(* CoDeSys 2.3.9.47 project: derevo_2016_12_28.pr6 *)
(* Author: Yurko Shybaigolova *)
(* Libraries: PlcHelperBC.lb6 7.5.01 11:03:00, TcAdsBC.lb6 5.7.02 11:03:02, standard.lb6 5.6.98 11:03:02, PlcSystemBC.lb6 21.3.01 11:03:02, TcBABasicBC.lb6 22.7.15 15:46:36, TcPlcUtilitiesBC.lb6 13.5.05 11:19:40 *)

(* Global variable list: main *)
VAR_GLOBAL
	data3floor: ARRAY[0..100] OF BYTE;
	data3floor_prev :ARRAY[0..100] OF BYTE;

	ads_adr1: STRING:='10.0.5.61.1.1';
	ads_adr2: STRING:='10.0.5.62.1.1';
	ads_adr3: STRING:='10.0.5.63.1.1';
	ads_adr_gym: STRING:='10.0.5.67.1.1';

	write_ads: ADSWRITE;
	basseinWindowToSafePos: BOOL;

	bDarkOutside		AT%MX0.0:BOOL;


	iHour			AT%MB4:BYTE;
	iMinute			AT%MB5:BYTE;
	lights			AT%MB6:DWORD;
	t_out			AT%MB10:INT;

	eib_vidpochynok1 				AT %MX100.0:	 BOOL;
	eib_vidpochynok2 				AT %MX100.1:	 BOOL;
	eib_veranda 					AT %MX100.2:	 BOOL;
	eib_veranda_zovn 				AT %MX100.3:	 BOOL;
	eib_vhid_zovn 					AT %MX100.4:	 BOOL;
	eib_sauna 						AT %MX100.5:	 BOOL;
	eib_vhid						AT %MX100.6:	 BOOL;
	eib_kotel 						AT %MX100.7:	 BOOL;

	eib_korydor 						AT %MX101.0:	 BOOL;
	eib_sinna 						AT %MX101.1:	 BOOL;
	eib_hamam 						AT %MX101.2:	 BOOL;
	eib_kuhnya 						AT %MX101.3:	 BOOL;
	eib_bassein1					AT %MX101.4:	 BOOL;
	eib_bassein_lampa				AT %MX101.5:	 BOOL;
	eib_spalnya2					AT %MX101.6:	 BOOL;
	eib_terassa 						AT %MX101.7:	 BOOL;

	eib_dush 						AT %MX102.0:	 BOOL;
	eib_wc 							AT %MX102.1:	 BOOL;
	eib_spalnya_verh				AT %MX102.2:	 BOOL;
	eib_spalnya1 					AT %MX102.3:	 BOOL;
	eib_spalnya_su 					AT %MX102.4:	 BOOL;
	eib_garderob 					AT %MX102.5:	 BOOL;
	eib_dush2						AT %MX102.6:	 BOOL;

	eib_okno_basseina				AT %MX103.0:	 BOOL;

	okno_basseina_status: BOOL;

	dataToGym0					AT %MB105: 	 BYTE;
	dataToGym1					AT %MB106: 	 BYTE;
	dataToGym2					AT %MB107: 	 BYTE;
	dataToGym3					AT %MB108: 	 BYTE;
	dataToGym4					AT %MB109: 	 BYTE;
	dataToGym5					AT %MB110: 	 BYTE;
	dataToGym6					AT %MB111: 	 BYTE;
	dataToGym7					AT %MB112: 	 BYTE;
	dataToGym8					AT %MB113: 	 BYTE;

	dataFromGym 				AT %MB300:	ARRAY[0..15] OF BYTE;





END_VAR

(* Global variable list: physical *)
(* @GLOBAL_VARIABLE_LIST := TwinCAT_Import *)
(* @PATH := '' *)
VAR_GLOBAL (* DO NOT CHANGE THIS SHEET MANUALLY! *)
	PlcInVar_0	AT %QB128:	USINT;
	PlcInVar_1	AT %QB129:	USINT;
	PlcInVar_2	AT %QB130:	USINT;
	PlcInVar_3	AT %QB131:	USINT;
	PlcInVar_4	AT %QB132:	USINT;
	PlcInVar_5	AT %QB133:	USINT;
	PlcInVar_6	AT %QB134:	USINT;
	PlcInVar_7	AT %QB135:	USINT;
	PlcInVar_8	AT %QB136:	USINT;
	PlcInVar_9	AT %QB137:	USINT;
	PlcInVar_10	AT %QB138:	USINT;
	PlcInVar_11	AT %QB139:	USINT;
	PlcInVar_12	AT %QB140:	USINT;
	PlcInVar_13	AT %QB141:	USINT;
	PlcInVar_14	AT %QB142:	USINT;
	PlcInVar_15	AT %QB143:	USINT;
	PlcOutVar_0	AT %IB128:	USINT;
	PlcOutVar_1	AT %IB129:	USINT;
	PlcOutVar_2	AT %IB130:	USINT;
	PlcOutVar_3	AT %IB131:	USINT;
	PlcOutVar_4	AT %IB132:	USINT;
	PlcOutVar_5	AT %IB133:	USINT;
	PlcOutVar_6	AT %IB134:	USINT;
	PlcOutVar_7	AT %IB135:	USINT;
	PlcOutVar_8	AT %IB136:	USINT;
	PlcOutVar_9	AT %IB137:	USINT;
	PlcOutVar_10	AT %IB138:	USINT;
	PlcOutVar_11	AT %IB139:	USINT;
	PlcOutVar_12	AT %IB140:	USINT;
	PlcOutVar_13	AT %IB141:	USINT;
	PlcOutVar_14	AT %IB142:	USINT;
	PlcOutVar_15	AT %IB143:	USINT;

	vidpochynok1	AT %QX0.0:	BOOL;
	vidpochynok2	AT %QX0.1:	BOOL;
	veranda 		AT %QX0.2:	BOOL;
	veranda_zovn	AT %QX0.3:	BOOL;
	vhid_zovn		AT %QX0.4:	BOOL;
	sauna			AT %QX0.5:	BOOL;
	vhid			AT %QX0.6:	BOOL;
(*c8*)kotel			AT %QX0.7:	BOOL;
	korydor			AT %QX1.0:	BOOL;
	sinna			AT %QX1.1:	BOOL;
	hamam			AT %QX1.2:	BOOL;
	kuhnya			AT %QX1.3:	BOOL;
	bassein1		AT %QX1.4:	BOOL;
	bassein2		AT %QX1.5:	BOOL;
	spalnya2		AT %QX1.6:	BOOL;
	terassa			AT %QX1.7:	BOOL;
	dush			AT %QX2.0:	BOOL;
	wc				AT %QX2.1:	BOOL;
	spalnya_verh	AT %QX2.2:	BOOL;
	spalnya1		AT %QX2.3:	BOOL;
	spalnya_su		AT %QX2.4:	BOOL;
	garderob		AT %QX2.5:	BOOL;
	Term_3_KL2408_7_Output	AT %QX2.6:	BOOL;
	Term_3_KL2408_8_Output	AT %QX2.7:	BOOL;

	dush2			AT %QX3.0:	BOOL;
	bassein_lampa	AT %QX3.1:	BOOL;
	bassein_okno_open	AT %QX3.2:	BOOL;
	bassein_okno_close AT %QX3.3:	BOOL;
	Term_4_KL2408_5_Output	AT %QX3.4:	BOOL;
	Term_4_KL2408_6_Output	AT %QX3.5:	BOOL;
	Term_4_KL2408_7_Output	AT %QX3.6:	BOOL;
	Term_4_KL2408_8_Output	AT %QX3.7:	BOOL;




	sw_vidpochynok1			AT %IX0.0:	BOOL;
	sw_vidpochynok2			AT %IX0.1:	BOOL;
	sw_veranda1				AT %IX0.2:	BOOL;
	sw_veranda2				AT %IX0.3:	BOOL;
	sw_spalnya1				AT %IX0.4:	BOOL;
	sw_spalnya2				AT %IX0.5:	BOOL;
	sw_vhid1			AT %IX0.6:	BOOL;
	sw_vhid2			AT %IX0.7:	BOOL;
	sw_korydor1				AT %IX1.0:	BOOL;
	sw_korydor2				AT %IX1.1:	BOOL;
	sw_vidpochynok_skhody1	AT %IX1.2:	BOOL;
	sw_vidpochynok_skhody2	AT %IX1.3:	BOOL;
	sw_sauna1				AT %IX1.4:	BOOL;
	sw_sauna2				AT %IX1.5:	BOOL;
	sw_bassein1				AT %IX1.6:	BOOL;
	sw_bassein2				AT %IX1.7:	BOOL;
	sw_sauna_vhid2		AT %IX2.0:	BOOL;
	sw_sauna_vhid1		AT %IX2.1:	BOOL;
	sw_sinna1					AT %IX2.2:	BOOL;
	Term_7_KL1408_4_Input	AT %IX2.3:	BOOL;
	sw_spalnya_su				AT %IX2.4:	BOOL;
	sw_garderob				AT %IX2.5:	BOOL;
	sw_kuh1					AT %IX2.6:	BOOL;
	sw_kuh2					AT %IX2.7:	BOOL;
	Term_8_KL1408_1_Input	AT %IX3.0:	BOOL;
	sw_sinna						AT %IX3.1:	BOOL;
	sw_skhody_22					AT %IX3.2:	BOOL;
	sw_skhody_21					AT %IX3.3:	BOOL;
	sw_skhody_12					AT %IX3.4:	BOOL;
	sw_skhody_11					AT %IX3.5:	BOOL;
	sw_hamam					AT %IX3.6:	BOOL;
	sw_spalnya_verh			AT %IX3.7:	BOOL;
	sw_terr1					AT %IX4.0:	BOOL;
	sw_terr2					AT %IX4.1:	BOOL;
	Term_9_KL1408_3_Input	AT %IX4.2:	BOOL;
	Term_9_KL1408_4_Input	AT %IX4.3:	BOOL;
	Term_9_KL1408_5_Input	AT %IX4.4:	BOOL;
	Term_9_KL1408_6_Input	AT %IX4.5:	BOOL;
	Term_9_KL1408_7_Input	AT %IX4.6:	BOOL;
	Term_9_KL1408_8_Input	AT %IX4.7:	BOOL;
END_VAR

(* @OBJECT_END := TwinCAT_Import *)

VAR_GLOBAL
END_VAR

(* POU MAIN, ST *)
PROGRAM MAIN
VAR
	i,j:INT;
	write:BOOL;
	heartBeat: TP;
	init:BOOL:=TRUE;

END_VAR
IF init THEN
	basseinWindowToSafePos:=TRUE;
	init:=FALSE;
END_IF

heartBeat(IN:= NOT heartBeat.Q, PT:=t#5s);

Light;


(*
IF NOT heartBeat.Q THEN
	knx_synchro;
END_IF
*)
write_data3floor;

ADS_Communication;

basseinWindowToSafePos:=FALSE;
END_PROGRAM
ACTION knx_synchro:
eib_vidpochynok1:=vidpochynok1;
eib_vidpochynok2 				:=vidpochynok2;
eib_veranda 					:=veranda;
eib_veranda_zovn 				:=veranda_zovn;
eib_vhid_zovn 					:=vhid_zovn;
eib_sauna 						:=sauna;
eib_vhid						:=vhid;
eib_kotel 						:=kotel;
eib_korydor 						:=korydor;
eib_sinna 						:=sinna;
eib_hamam 						:=hamam;
eib_kuhnya 						:=kuhnya;
eib_bassein1					:=bassein1;
eib_bassein_lampa				:=bassein_lampa;
eib_spalnya2					:=spalnya2;
eib_terassa 						:=terassa;
eib_dush 						:=dush;
eib_wc 							:=wc;
eib_spalnya_verh				:=spalnya_verh;
eib_spalnya1 					:=spalnya1;
eib_spalnya_su 					:=spalnya_su;
eib_garderob 					:=garderob;
eib_dush2						:=dush2;
END_ACTION
ACTION write_data3floor:
	data3floor[0].0:= vidpochynok1 ;
	data3floor[0].1:= vidpochynok2 ;
	data3floor[0].2:= veranda ;
	data3floor[0].3:= veranda_zovn ;
	data3floor[0].4:= vhid_zovn ;
	data3floor[0].5:= sauna ;
	data3floor[0].6:= vhid	;
	data3floor[0].7:= kotel;

	data3floor[1].0:= korydor ;
	data3floor[1].1:= sinna ;
	data3floor[1].2:= hamam ;
	data3floor[1].3:= kuhnya ;
	data3floor[1].4:= bassein1	;
	data3floor[1].5:= bassein_lampa;
	data3floor[1].6:= spalnya2;
	data3floor[1].7:= terassa;

	data3floor[2].0:= dush ;
	data3floor[2].1:= wc ;
	data3floor[2].2:= spalnya_verh	;
	data3floor[2].3:= spalnya1 ;
	data3floor[2].4:= spalnya_su ;
	data3floor[2].5:= garderob ;
	data3floor[2].6:= dush2;

	data3floor[3].0:= okno_basseina_status;

MEMCPY( destAddr := ADR( data3floor[10] ), srcAddr := ADR(dataFromGym), n := SIZEOF( dataFromGym) );

FOR i:=0 TO (SIZEOF(data3floor))-1 DO
	IF data3floor[i]<>data3floor_prev[i]  THEN
		write:=TRUE;
		EXIT;
	ELSE
		write:=FALSE;
	END_IF
END_FOR


FOR j:=0 TO (SIZEOF(data3floor))-1 DO
	data3floor_prev[j]:=data3floor[j];
END_FOR
END_ACTION

(* POU lights/Light, CFC *)
PROGRAM Light
VAR
	fbLight_vidpochynok1: fb_light;
	fbLight_vidpochynok2: fb_light;
	fbLight_veranda: fb_light;
	fbLight_veranda_zovn: fb_light;
	fbLight_vhid_zovn: fb_light;
	fbLight_sauna: FB_Light;
	fbLight_vhid: fb_light;
	fbLight_kotel: fb_light;
	fbLight_korydor: fb_light;
	fbLight_sinna: FB_Light;
	fbLight_hamam: fb_light;
	fbLight_kuhnya: fb_light;
	fbLight_bassein1: FB_Light;
	fbLight_bassein_lampa: FB_Light;
	fbLight_spalnya2: fb_light;
	fbLight_terassa: fb_light;
	fbLight_dush: fb_light;
	fbLight_wc: fb_light;
	fbLight_spalnya_verh: FB_Light;
	fbLight_spalnya1: fb_light;
	fbLight_spalnya_su: FB_Light;
	fbLight_garderob: FB_Light;
	fbLight_spalnya_verkh: FB_Light;
	fbLight_kuhnya_pidsvitka: FB_Light;
	R_polka: R_TRIG;
	F_polka: F_TRIG;
	fb_swKorydor2: FB_ShortLongClick;
	fb_swBassein2: FB_ShortLongClick;
	fb_swKorydor1: FB_ShortLongClick;
	fbLight_dush2: FB_Light;
	fbBasseinWindow: FB_RoofWindow;
	fbBasseinWindowCtrl: FB_Light;

	okno_basseina_status_SET_RESET: SEMA;
END_VAR
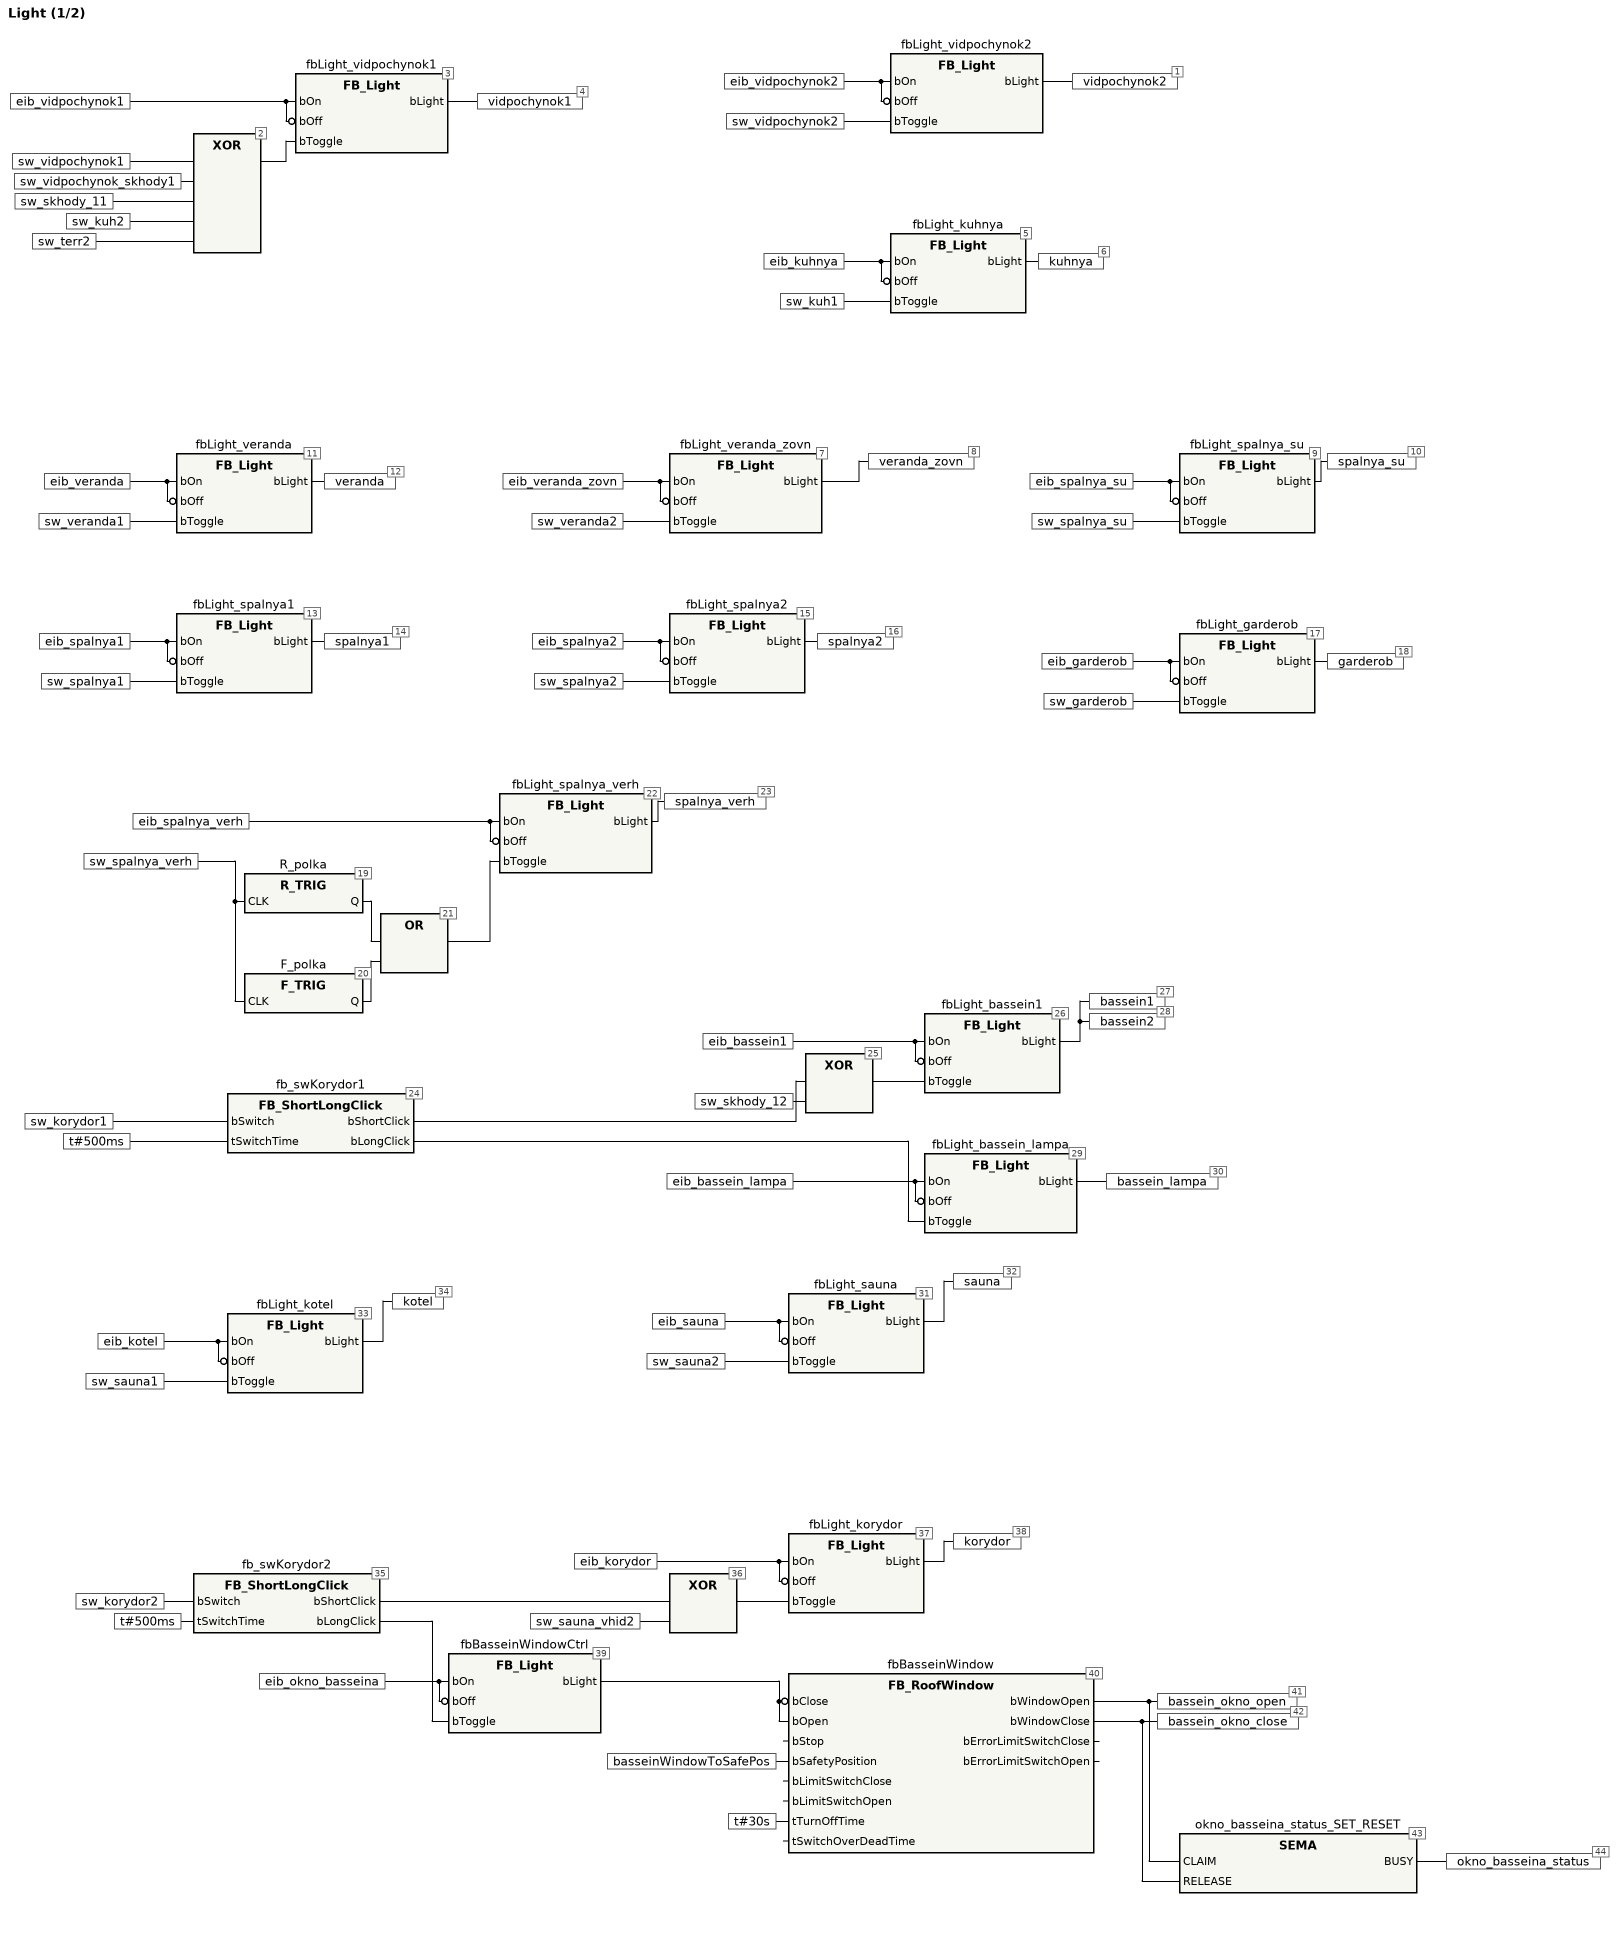
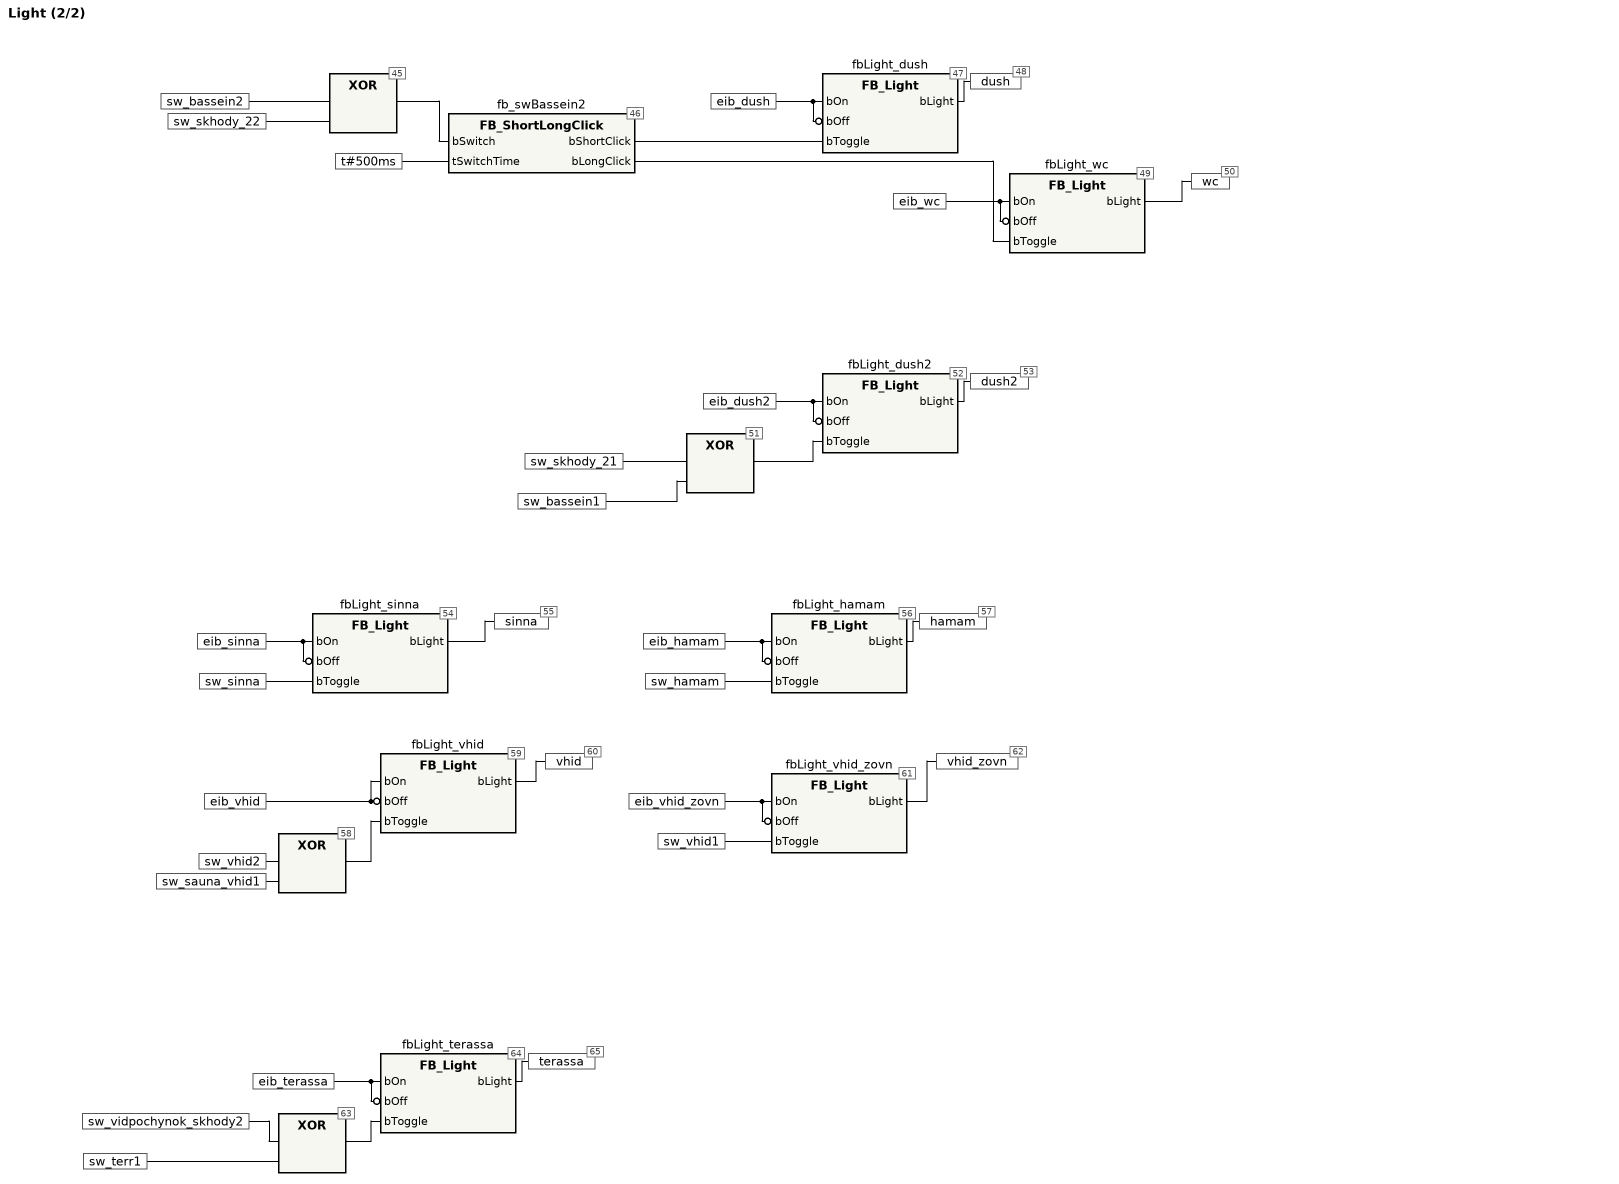
_CFC_ (* Continuous Function Chart, elements in execution order *)
#0 fbLight_vidpochynok2:FB_Light(bOn: eib_vidpochynok2, bOff: NOT eib_vidpochynok2, bToggle: sw_vidpochynok2)
#1 vidpochynok2 <= #0.bLight
#2 XOR(sw_vidpochynok1, sw_vidpochynok_skhody1, sw_skhody_11, sw_kuh2, sw_terr2)
#3 fbLight_vidpochynok1:FB_Light(bOn: eib_vidpochynok1, bOff: NOT eib_vidpochynok1, bToggle: #2)
#4 vidpochynok1 <= #3.bLight
#5 fbLight_kuhnya:FB_Light(bOn: eib_kuhnya, bOff: NOT eib_kuhnya, bToggle: sw_kuh1)
#6 kuhnya <= #5.bLight
#7 fbLight_veranda_zovn:FB_Light(bOn: eib_veranda_zovn, bOff: NOT eib_veranda_zovn, bToggle: sw_veranda2)
#8 veranda_zovn <= #7.bLight
#9 fbLight_spalnya_su:FB_Light(bOn: eib_spalnya_su, bOff: NOT eib_spalnya_su, bToggle: sw_spalnya_su)
#10 spalnya_su <= #9.bLight
#11 fbLight_veranda:FB_Light(bOn: eib_veranda, bOff: NOT eib_veranda, bToggle: sw_veranda1)
#12 veranda <= #11.bLight
#13 fbLight_spalnya1:FB_Light(bOn: eib_spalnya1, bOff: NOT eib_spalnya1, bToggle: sw_spalnya1)
#14 spalnya1 <= #13.bLight
#15 fbLight_spalnya2:FB_Light(bOn: eib_spalnya2, bOff: NOT eib_spalnya2, bToggle: sw_spalnya2)
#16 spalnya2 <= #15.bLight
#17 fbLight_garderob:FB_Light(bOn: eib_garderob, bOff: NOT eib_garderob, bToggle: sw_garderob)
#18 garderob <= #17.bLight
#19 R_polka:R_TRIG(CLK: sw_spalnya_verh)
#20 F_polka:F_TRIG(CLK: sw_spalnya_verh)
#21 OR(#19.Q, #20.Q)
#22 fbLight_spalnya_verh:FB_Light(bOn: eib_spalnya_verh, bOff: NOT eib_spalnya_verh, bToggle: #21)
#23 spalnya_verh <= #22.bLight
#24 fb_swKorydor1:FB_ShortLongClick(bSwitch: sw_korydor1, tSwitchTime: t#500ms)
#25 XOR(#24.bShortClick, sw_skhody_12)
#26 fbLight_bassein1:FB_Light(bOn: eib_bassein1, bOff: NOT eib_bassein1, bToggle: #25)
#27 bassein1 <= #26.bLight
#28 bassein2 <= #26.bLight
#29 fbLight_bassein_lampa:FB_Light(bOn: eib_bassein_lampa, bOff: NOT eib_bassein_lampa, bToggle: #24.bLongClick)
#30 bassein_lampa <= #29.bLight
#31 fbLight_sauna:FB_Light(bOn: eib_sauna, bOff: NOT eib_sauna, bToggle: sw_sauna2)
#32 sauna <= #31.bLight
#33 fbLight_kotel:FB_Light(bOn: eib_kotel, bOff: NOT eib_kotel, bToggle: sw_sauna1)
#34 kotel <= #33.bLight
#35 fb_swKorydor2:FB_ShortLongClick(bSwitch: sw_korydor2, tSwitchTime: t#500ms)
#36 XOR(#35.bShortClick, sw_sauna_vhid2)
#37 fbLight_korydor:FB_Light(bOn: eib_korydor, bOff: NOT eib_korydor, bToggle: #36)
#38 korydor <= #37.bLight
#39 fbBasseinWindowCtrl:FB_Light(bOn: eib_okno_basseina, bOff: NOT eib_okno_basseina, bToggle: #35.bLongClick)
#40 fbBasseinWindow:FB_RoofWindow(bClose: NOT #39.bLight, bOpen: #39.bLight, bStop: -, bSafetyPosition: basseinWindowToSafePos, bLimitSwitchClose: -, bLimitSwitchOpen: -, tTurnOffTime: t#30s, tSwitchOverDeadTime: -)
#41 bassein_okno_open <= #40.bWindowOpen
#42 bassein_okno_close <= #40.bWindowClose
#43 okno_basseina_status_SET_RESET:SEMA(CLAIM: #40.bWindowOpen, RELEASE: #40.bWindowClose)
#44 okno_basseina_status <= #43.BUSY
#45 XOR(sw_bassein2, sw_skhody_22)
#46 fb_swBassein2:FB_ShortLongClick(bSwitch: #45, tSwitchTime: t#500ms)
#47 fbLight_dush:FB_Light(bOn: eib_dush, bOff: NOT eib_dush, bToggle: #46.bShortClick)
#48 dush <= #47.bLight
#49 fbLight_wc:FB_Light(bOn: eib_wc, bOff: NOT eib_wc, bToggle: #46.bLongClick)
#50 wc <= #49.bLight
#51 XOR(sw_skhody_21, sw_bassein1)
#52 fbLight_dush2:FB_Light(bOn: eib_dush2, bOff: NOT eib_dush2, bToggle: #51)
#53 dush2 <= #52.bLight
#54 fbLight_sinna:FB_Light(bOn: eib_sinna, bOff: NOT eib_sinna, bToggle: sw_sinna)
#55 sinna <= #54.bLight
#56 fbLight_hamam:FB_Light(bOn: eib_hamam, bOff: NOT eib_hamam, bToggle: sw_hamam)
#57 hamam <= #56.bLight
#58 XOR(sw_vhid2, sw_sauna_vhid1)
#59 fbLight_vhid:FB_Light(bOn: eib_vhid, bOff: NOT eib_vhid, bToggle: #58)
#60 vhid <= #59.bLight
#61 fbLight_vhid_zovn:FB_Light(bOn: eib_vhid_zovn, bOff: NOT eib_vhid_zovn, bToggle: sw_vhid1)
#62 vhid_zovn <= #61.bLight
#63 XOR(sw_vidpochynok_skhody2, sw_terr1)
#64 fbLight_terassa:FB_Light(bOn: eib_terassa, bOff: NOT eib_terassa, bToggle: #63)
#65 terassa <= #64.bLight
_END_CFC_
(* the same logic as Structured Text *)
fbLight_vidpochynok2(bOn := eib_vidpochynok2, bOff := NOT eib_vidpochynok2, bToggle := sw_vidpochynok2);
vidpochynok2 := fbLight_vidpochynok2.bLight;
fbLight_vidpochynok1(bOn := eib_vidpochynok1, bOff := NOT eib_vidpochynok1, bToggle := sw_vidpochynok1 XOR sw_vidpochynok_skhody1 XOR sw_skhody_11 XOR sw_kuh2 XOR sw_terr2);
vidpochynok1 := fbLight_vidpochynok1.bLight;
fbLight_kuhnya(bOn := eib_kuhnya, bOff := NOT eib_kuhnya, bToggle := sw_kuh1);
kuhnya := fbLight_kuhnya.bLight;
fbLight_veranda_zovn(bOn := eib_veranda_zovn, bOff := NOT eib_veranda_zovn, bToggle := sw_veranda2);
veranda_zovn := fbLight_veranda_zovn.bLight;
fbLight_spalnya_su(bOn := eib_spalnya_su, bOff := NOT eib_spalnya_su, bToggle := sw_spalnya_su);
spalnya_su := fbLight_spalnya_su.bLight;
fbLight_veranda(bOn := eib_veranda, bOff := NOT eib_veranda, bToggle := sw_veranda1);
veranda := fbLight_veranda.bLight;
fbLight_spalnya1(bOn := eib_spalnya1, bOff := NOT eib_spalnya1, bToggle := sw_spalnya1);
spalnya1 := fbLight_spalnya1.bLight;
fbLight_spalnya2(bOn := eib_spalnya2, bOff := NOT eib_spalnya2, bToggle := sw_spalnya2);
spalnya2 := fbLight_spalnya2.bLight;
fbLight_garderob(bOn := eib_garderob, bOff := NOT eib_garderob, bToggle := sw_garderob);
garderob := fbLight_garderob.bLight;
R_polka(CLK := sw_spalnya_verh);
F_polka(CLK := sw_spalnya_verh);
fbLight_spalnya_verh(bOn := eib_spalnya_verh, bOff := NOT eib_spalnya_verh, bToggle := R_polka.Q OR F_polka.Q);
spalnya_verh := fbLight_spalnya_verh.bLight;
fb_swKorydor1(bSwitch := sw_korydor1, tSwitchTime := t#500ms);
fbLight_bassein1(bOn := eib_bassein1, bOff := NOT eib_bassein1, bToggle := fb_swKorydor1.bShortClick XOR sw_skhody_12);
bassein1 := fbLight_bassein1.bLight;
bassein2 := fbLight_bassein1.bLight;
fbLight_bassein_lampa(bOn := eib_bassein_lampa, bOff := NOT eib_bassein_lampa, bToggle := fb_swKorydor1.bLongClick);
bassein_lampa := fbLight_bassein_lampa.bLight;
fbLight_sauna(bOn := eib_sauna, bOff := NOT eib_sauna, bToggle := sw_sauna2);
sauna := fbLight_sauna.bLight;
fbLight_kotel(bOn := eib_kotel, bOff := NOT eib_kotel, bToggle := sw_sauna1);
kotel := fbLight_kotel.bLight;
fb_swKorydor2(bSwitch := sw_korydor2, tSwitchTime := t#500ms);
fbLight_korydor(bOn := eib_korydor, bOff := NOT eib_korydor, bToggle := fb_swKorydor2.bShortClick XOR sw_sauna_vhid2);
korydor := fbLight_korydor.bLight;
fbBasseinWindowCtrl(bOn := eib_okno_basseina, bOff := NOT eib_okno_basseina, bToggle := fb_swKorydor2.bLongClick);
fbBasseinWindow(bClose := NOT fbBasseinWindowCtrl.bLight, bOpen := fbBasseinWindowCtrl.bLight, bSafetyPosition := basseinWindowToSafePos, tTurnOffTime := t#30s);
bassein_okno_open := fbBasseinWindow.bWindowOpen;
bassein_okno_close := fbBasseinWindow.bWindowClose;
okno_basseina_status_SET_RESET(CLAIM := fbBasseinWindow.bWindowOpen, RELEASE := fbBasseinWindow.bWindowClose);
okno_basseina_status := okno_basseina_status_SET_RESET.BUSY;
fb_swBassein2(bSwitch := sw_bassein2 XOR sw_skhody_22, tSwitchTime := t#500ms);
fbLight_dush(bOn := eib_dush, bOff := NOT eib_dush, bToggle := fb_swBassein2.bShortClick);
dush := fbLight_dush.bLight;
fbLight_wc(bOn := eib_wc, bOff := NOT eib_wc, bToggle := fb_swBassein2.bLongClick);
wc := fbLight_wc.bLight;
fbLight_dush2(bOn := eib_dush2, bOff := NOT eib_dush2, bToggle := sw_skhody_21 XOR sw_bassein1);
dush2 := fbLight_dush2.bLight;
fbLight_sinna(bOn := eib_sinna, bOff := NOT eib_sinna, bToggle := sw_sinna);
sinna := fbLight_sinna.bLight;
fbLight_hamam(bOn := eib_hamam, bOff := NOT eib_hamam, bToggle := sw_hamam);
hamam := fbLight_hamam.bLight;
fbLight_vhid(bOn := eib_vhid, bOff := NOT eib_vhid, bToggle := sw_vhid2 XOR sw_sauna_vhid1);
vhid := fbLight_vhid.bLight;
fbLight_vhid_zovn(bOn := eib_vhid_zovn, bOff := NOT eib_vhid_zovn, bToggle := sw_vhid1);
vhid_zovn := fbLight_vhid_zovn.bLight;
fbLight_terassa(bOn := eib_terassa, bOff := NOT eib_terassa, bToggle := sw_vidpochynok_skhody2 XOR sw_terr1);
terassa := fbLight_terassa.bLight;
END_PROGRAM

(* POU ADS_Communication, CFC *)
PROGRAM ADS_Communication
VAR
	fb_floor3ADSwrite: ADSWRITE;
	fb_GymADSwrite: ADSWRITE;


	counter_error,counter_busy: CTU;
END_VAR
VAR (* helpers for the ST form of the networks *)
	_t21 : DWORD;
	_t23 : DWORD;
	_t42 : BOOL;
	_t56 : DWORD;
	_t60 : BOOL;
END_VAR
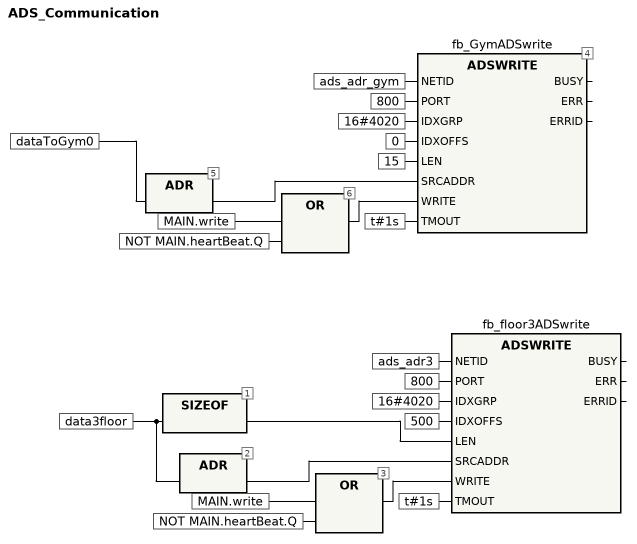
_CFC_ (* Continuous Function Chart, elements in execution order *)
#0 fb_floor3ADSwrite:ADSWRITE(NETID: ads_adr3, PORT: 800, IDXGRP: 16#4020, IDXOFFS: 500, LEN: #1, SRCADDR: #2, WRITE: #3, TMOUT: t#1s)
#1 SIZEOF(data3floor)
#2 ADR(data3floor)
#3 OR(MAIN.write, NOT MAIN.heartBeat.Q)
#4 fb_GymADSwrite:ADSWRITE(NETID: ads_adr_gym, PORT: 800, IDXGRP: 16#4020, IDXOFFS: 0, LEN: 15, SRCADDR: #5, WRITE: #6, TMOUT: t#1s)
#5 ADR(dataToGym0)
#6 OR(MAIN.write, NOT MAIN.heartBeat.Q)
_END_CFC_
(* the same logic as Structured Text *)
fb_floor3ADSwrite(NETID := ads_adr3, PORT := 800, IDXGRP := 16#4020, IDXOFFS := 500, LEN := _t21, SRCADDR := _t23, WRITE := _t42, TMOUT := t#1s);
_t21 := SIZEOF(data3floor);
_t23 := ADR(data3floor);
_t42 := MAIN.write OR NOT MAIN.heartBeat.Q;
fb_GymADSwrite(NETID := ads_adr_gym, PORT := 800, IDXGRP := 16#4020, IDXOFFS := 0, LEN := 15, SRCADDR := _t56, WRITE := _t60, TMOUT := t#1s);
_t56 := ADR(dataToGym0);
_t60 := MAIN.write OR NOT MAIN.heartBeat.Q;
END_PROGRAM

(* POU ADS_write, ST *)
PROGRAM ADS_write
VAR
	write_timeout: TIME;
	b_write3, b_write2: BOOL;
	write_ads3, write_ads2: ADSWRITE;

	timer3, timer2:TP;
	errorcounter3, errorcounter2, pack_c:CTU ;
	test_word: WORD;
	i,j,i1,j1: INT;
	data_changed: BOOL;
	try_again2, try_again3: BOOL;
	temp: INT;
	SENT2, SENT3:F_TRIG;
	SNT_CNT2, SNT_CNT3:CTU;
	fb_heartbeat_timer: TON;
END_VAR
write_data3floor;
write_timeout:=t#1s;
fb_heartbeat_timer(in:=NOT fb_heartbeat_timer.Q, pt:=t#10s);

(*3floor*)
FOR i1:=0 TO (SIZEOF(data3floor)-1)-1DO
	IF data3floor[i1]<>data3floor_prev[i1] OR fb_heartbeat_timer.Q  THEN
		b_write3:=TRUE;
		EXIT;
	ELSE
		b_write3:=FALSE;
	END_IF
END_FOR

IF try_again3 AND NOT timer3.Q THEN
	b_write3:=TRUE;
	try_again3:=FALSE;
END_IF


IF write_ads3.BUSY THEN b_write3:=FALSE; END_IF

	write_ads3(
		NETID:=ads_adr3,
		PORT:=801,
		IDXGRP:=16#4020,
		IDXOFFS:=400,
		WRITE:=b_write3,
		TMOUT:=write_timeout,
		LEN:=SIZEOF(data3floor),
		SRCADDR:=ADR(data3floor));

IF write_ads3.ERR AND NOT timer3.Q THEN
	timer3.IN:=TRUE;
	try_again3:=TRUE;
END_IF
timer3(PT:=write_timeout);
timer3.IN:=FALSE;

SENT3(CLK:=write_ads3.BUSY);

IF NOT write_ads3.ERR THEN
	SNT_CNT3(CU:=SENT3.Q);
END_IF

FOR j1:=0 TO (SIZEOF(data3floor)-1)-1 DO
	data3floor_prev[j1]:=data3floor[j1];
END_FOR
END_PROGRAM

(* POU lights/fbMoovingSensorLight, ST *)
FUNCTION_BLOCK fbMoovingSensorLight
VAR_INPUT
	button:BOOL;
	duration:TIME;
	sensor:BOOL;
	knx:BOOL;
END_VAR
VAR_OUTPUT
	out: BOOL;
END_VAR
VAR
	fbStairwayLight_00			: FB_StairwellLight;
	button_rising				: R_TRIG;
	sensor_falling				: F_TRIG;
	timer_falling					: F_TRIG;
	knx_falling					: F_TRIG;
	knx_rising					: R_TRIG;
END_VAR

VAR_IN_OUT
END_VAR
knx_rising(CLK:=knx);
knx_falling(CLK:=knx);
button_rising(CLK:=button);
sensor_falling(CLK:= sensor);
timer_falling(clk:=fbStairwayLight_00.bStart);

IF sensor_falling.Q AND NOT out THEN
	fbStairwayLight_00.bOff:=FALSE;
END_IF

fbStairwayLight_00(
	bSwitch:=NOT sensor AND NOT out,
	tLightDuration:=duration,
	tPreWarningStart:=t#100s,
	tPreWarningDuration:=t#500ms);

IF fbStairwayLight_00.bStart THEN
	out := fbStairwayLight_00.bLight;
END_IF

IF timer_falling.Q THEN
	out:=FALSE;
END_IF




IF knx_rising.Q OR knx_falling.Q THEN
	out:= knx;
	IF knx_falling.Q THEN
		fbStairwayLight_00.bOff:=TRUE;
	END_IF
END_IF

IF button_rising.Q THEN
	out:= NOT out;
	fbStairwayLight_00.bOff:=TRUE;
END_IF
END_FUNCTION_BLOCK
